FUNCTION_BLOCK FB_UnixTimestamp
VAR_OUTPUT
    seconds: ULINT;
//    milliseconds: ULINT;
END_VAR

VAR
    localSystemTime : FB_LocalSystemTime := ( bEnable := TRUE, dwCycle := 1 );
    getTimeZoneInformation : FB_GetTimeZoneInformation;
    timeZoneInformation : ST_TimeZoneInformation;
    specificLocalTimeToFileTime : FB_TzSpecificLocalTimeToFileTime;
    fileTime: T_FILETIME;
    onZerothSecondLastCycle : BOOL;
END_VAR

// Get local system time
localSystemTime();

// On the zeroth second of each minutesync timezone information
IF (timeZoneInformation.standardName = '' OR (localSystemTime.systemTime.wSecond = 0 AND NOT onZerothSecondLastCycle)) THEN
    getTimeZoneInformation(sNetID := '', bExecute := TRUE, tzInfo => timeZoneInformation);
END_IF;

// Convert local system time to unix timestamps
specificLocalTimeToFileTime(in := Tc2_Utilities.SYSTEMTIME_TO_FILETIME(localSystemTime.systemTime), tzInfo := timeZoneInformation, out => fileTime);
seconds := (SHL(DWORD_TO_ULINT(fileTime.dwHighDateTime), 32) + DWORD_TO_ULINT(fileTime.dwLowDateTime)) / 10000000 - 11644473600;
//milliseconds := (SHL(DWORD_TO_ULINT(fileTime.dwHighDateTime), 32) + DWORD_TO_ULINT(fileTime.dwLowDateTime)) / 10000 - 11644473600000;

onZerothSecondLastCycle := localSystemTime.systemTime.wSecond = 0;

END_FUNCTION_BLOCK

(* stored: Version 1.1.0.1, ProductVersion 3.1.4024.12
   POU FB_UnixTimestamp: Id {03fc0b33-257a-4e05-a053-22964feb09e5}, SpecialFunc None *)
